{attribute 'linkalways'} 
{attribute 'no_explicit_call' := 'This FB is a CLASS and must be accessed using methods or properties'}
{attribute 'enable_dynamic_creation'}
FUNCTION_BLOCK FINAL GT_UINT EXTENDS Node
VAR
	in1 : _UINT(0);
	in2 : _UINT(0);
	out : _BOOL(FALSE);
END_VAR

METHOD PUBLIC Clone : I_Node
VAR
	pNode : POINTER TO GT_UINT;
END_VAR
pNode := __NEW(GT_UINT);
Clone := pNode^;
END_METHOD

METHOD FB_init : BOOL
VAR_INPUT
	bInitRetains : BOOL; // if TRUE, the retain variables are initialized (warm start / cold start)
	bInCopyCode : BOOL;  // if TRUE, the instance afterwards gets moved into the copy code (online change)
END_VAR
AddInput('in1',THIS^.in1);
AddInput('in2',THIS^.in2);
AddOutput('out', THIS^.out);
END_METHOD

METHOD PROTECTED OnExecute
VAR
END_VAR
out.Value := in1.Value > in2.Value;
END_METHOD

END_FUNCTION_BLOCK

(* stored: Version 1.1.0.1, ProductVersion 3.1.4024.15
   POU GT_UINT: Id {49689906-4657-4f16-8729-71a4fc07068a}, SpecialFunc None
   Folder Constructor: Id {ab6eea99-4c12-4e48-acc7-c187975a178a}
   Method Clone: Id {7a732cb9-5ac4-4663-8cc1-2c784ade86d8}
   Method FB_init: Id {b309a157-77d9-42c9-b7a1-e4f685e88ec8}
   Method OnExecute: Id {9ff87130-8046-49c8-b2da-e29e8ef044e2} *)
